// Mitsubishi GX Works2 project: MOV_ROL   PLC: Q03UDV

PROGRAM MAIN
VAR
  PB1 : BOOL;
END_VAR
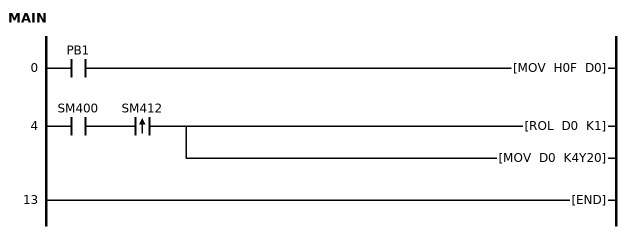
0     LD      PB1
      MOV     H0F D0
4     LD      SM400
      ANDP    SM412
      ROL     D0 K1
      MOV     D0 K4Y20
13    END
END_PROGRAM

PROGRAM MAIN1
0     END
END_PROGRAM
